// TIA Portal project "ASENKRON MOTORA YILDIZ UCGEN YOL VERME" (V18)

(* hardware
DEVICE "S7-1200 station_1"  S7-1200 Station
   slot 0: "Rack_0"  S7-1200 Rack  Rack  V1.0
   slot 1: "PLC_1"  CPU 1212C DC/DC/DC  6ES7 212-1AE40-0XB0  V4.6
*)

// ===== PLC "PLC_1"  CPU 1212C DC/DC/DC =====

VAR_GLOBAL   // PLC tag table "Default tag table"
   "START BUT" AT %I0.0 : Bool;
   "STOP BUT" AT %I0.1 : Bool;
   "ANA KONTAKTOR" AT %Q0.0 : Bool;
   "YILDIZ KONTAKTOR" AT %Q0.1 : Bool;
   "UCGEN KONTAKTOR" AT %Q0.2 : Bool;
END_VAR

// folder: System blocks/Program resources

DATA_BLOCK "TIMER"   // DB1
{ S7_Optimized_Access := 'TRUE' }
AUTHOR : Simatic
FAMILY : IEC
NAME : IEC_TMR
VERSION : 1.0
// stored: InstanceOfName IEC_TIMER
"IEC_TIMER"
BEGIN
END_DATA_BLOCK

// folder: (top level)

ORGANIZATION_BLOCK "Main"   // OB1, LAD, ProgramCycle
TITLE = "Main Program Sweep (Cycle)"
{ S7_Optimized_Access := 'TRUE' }
VERSION : 0.1
   VAR_INPUT
      Initial_Call : Bool;   // Initial call of this OB
      Remanence : Bool;   // =True, if remanent data are available
   END_VAR
BEGIN

REGION Network 1: SISTEM HAZIR
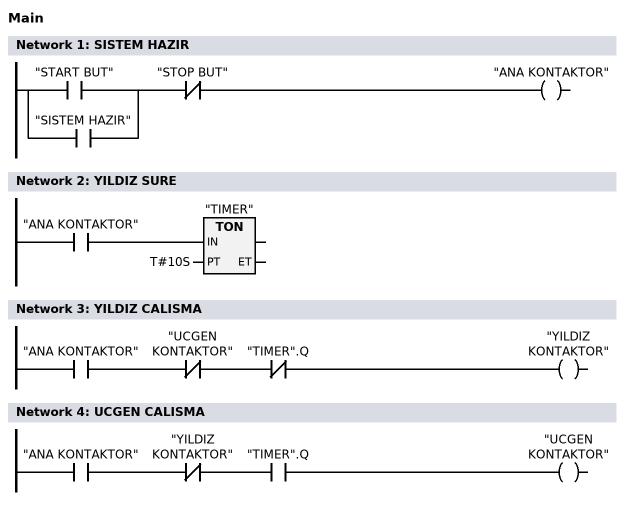
   RUNG wire#powerrail
      Contact( "START BUT" )
      wire#w1
      I_Contact( "STOP BUT" )
      Coil( "ANA KONTAKTOR" )
   END_RUNG
   RUNG wire#powerrail
      Contact( "SISTEM HAZIR" )
   END_RUNG wire#w1
   // the same network as SCL:
   "ANA KONTAKTOR" := ("START BUT" OR "SISTEM HAZIR") AND NOT "STOP BUT";
END_REGION

REGION Network 2: YILDIZ SURE
   "TIMER".TON(IN := "ANA KONTAKTOR", PT := T#10S);
END_REGION

REGION Network 3: YILDIZ CALISMA
   RUNG wire#powerrail
      Contact( "ANA KONTAKTOR" )
      I_Contact( "UCGEN KONTAKTOR" )
      I_Contact( "TIMER".Q )
      Coil( "YILDIZ KONTAKTOR" )
   END_RUNG
   // the same network as SCL:
   "YILDIZ KONTAKTOR" := "ANA KONTAKTOR" AND NOT "UCGEN KONTAKTOR" AND NOT "TIMER".Q;
END_REGION

REGION Network 4: UCGEN CALISMA
   RUNG wire#powerrail
      Contact( "ANA KONTAKTOR" )
      I_Contact( "YILDIZ KONTAKTOR" )
      Contact( "TIMER".Q )
      Coil( "UCGEN KONTAKTOR" )
   END_RUNG
   // the same network as SCL:
   "UCGEN KONTAKTOR" := "ANA KONTAKTOR" AND NOT "YILDIZ KONTAKTOR" AND "TIMER".Q;
END_REGION
END_ORGANIZATION_BLOCK